// Mitsubishi GX Works2 project: 14-06-2020 LAB 2_Sequence   PLC: FX3G

PROGRAM MAIN
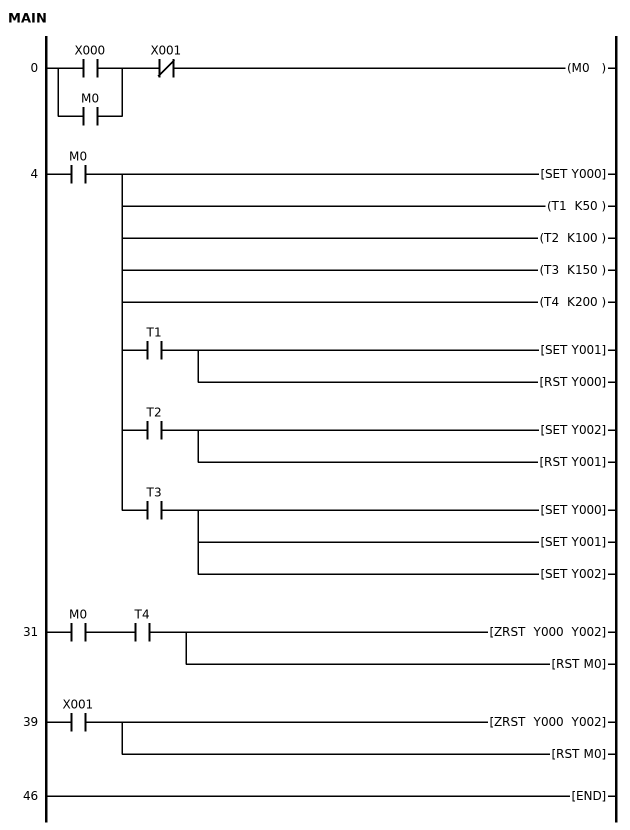
0     LD      X000
      OR      M0
      ANI     X001
      OUT     M0
4     LD      M0
      SET     Y000
      OUT     T1 K50
      OUT     T2 K100
      OUT     T3 K150
      OUT     T4 K200
      MPS
      AND     T1
      SET     Y001
      RST     Y000
      MRD
      AND     T2
      SET     Y002
      RST     Y001
      MPP
      AND     T3
      SET     Y000
      SET     Y001
      SET     Y002
31    LD      M0
      AND     T4
      ZRST    Y000 Y002
      RST     M0
39    LD      X001
      ZRST    Y000 Y002
      RST     M0
46    END
END_PROGRAM
